FUNCTION_BLOCK F_DIV (* Divides two values *)
  (* Standard: 61131-3; Classification: Mathematic; Function: DIVIDER; Type: Mathematical function *)
  (* Version 1.0, 2011-09-20, 4DIAC-IDE, 4DIAC-Consortium *)
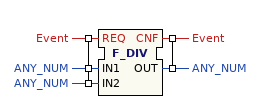
  EVENT_INPUT
    REQ WITH IN1, IN2; (* Normal Execution Request *)
  END_EVENT
  EVENT_OUTPUT
    CNF WITH OUT; (* Execution Confirmation *)
  END_EVENT
  VAR_INPUT
    IN1 : ANY_NUM; (* First funtion input *)
    IN2 : ANY_NUM; (* Second function input *)
  END_VAR
  VAR_OUTPUT
    OUT : ANY_NUM; (* Function output *)
  END_VAR
END_FUNCTION_BLOCK
